// Brief: Slave Arm Run Self-check Trajectory
FUNCTION_BLOCK PUBLIC FB_SlaveCtrlInstruRetract EXTENDS FB_SlaveArmCtrlBase
VAR_INPUT
END_VAR
VAR_OUTPUT
END_VAR
VAR
	m_retractPlanner:FB_BasicDoubleS;;
	
	m_retractVel: LREAL:= 0.05;
	m_retractAcc: LREAL:= 0.1;
	m_retractJerk: LREAL:= 1;
	
	m_retractLimitBuffer:LREAL := 0.02;
	m_retractPos :LREAL;
	
END_VAR

// override this function in each exact controller
METHOD PROTECTED calcCmdJntPos : BOOL
VAR_IN_OUT CONSTANT
	i_endoscopePose : ST_Frame;
	i_masterStatus :ST_MasterStatus;
	i_setupStatus: ST_SetupStatus;
	i_slaveArm :FB_SlaveArm;
END_VAR

VAR 
	i :INT;
	curJntVel :Vec8d;
END_VAR
// check if planner is ready
IF m_retractPlanner.isGene = FALSE THEN
	calcCmdJntPos:=FALSE;
	m_timePeriod:=0;
	RETURN;
END_IF

// traj plan
calcCmdJntPos :=m_retractPlanner.evaluate(m_timePeriod, q=> m_cmdJntPos[3], q_dot=>m_cmdJntVel[3], q_dot=> m_cmdJntAcc[3]);

IF m_timePeriod > m_retractPlanner.duration AND  ABS(i_slaveArm.curJntPos[3] - m_retractPos) < g_cartCtrlPosTolHign THEN
	m_isFinished:=TRUE;
END_IF
END_METHOD

METHOD PUBLIC init : BOOL
VAR_IN_OUT CONSTANT
	i_slaveArm	:FB_SlaveArm;
END_VAR
VAR_IN_OUT 
	r_slaveArmCtrlCmd :ST_SlaveArmCtrlCmds;
END_VAR

VAR
	q:ARRAY[1..2] OF LREAL;
	v:ARRAY[1..2] OF LREAL;
END_VAR
// check if to hold the command joint position unchanged
m_holdLastCmds := checkToHoldLastCmds(i_slaveArm);

SUPER^.Init(i_slaveArm,r_slaveArmCtrlCmd);

// planning for joint3 motion
m_retractPos :=GVL_SlaveMotorParameters.g_maxJntPos[3]+m_retractLimitBuffer;
q[1]:=i_slaveArm.curJntPos[3];
q[2]:= m_retractPos;
v[1]:=0;
v[2]:=0;
m_retractPlanner.init(q,v, m_retractVel, m_retractAcc, m_retractJerk);
END_METHOD

END_FUNCTION_BLOCK

(* stored: Version 1.1.0.1, ProductVersion 3.1.4024.11
   POU FB_SlaveCtrlInstruRetract: Id {596332da-68eb-4244-8a80-7e3d57b3bb9f}, SpecialFunc None
   Method calcCmdJntPos: Id {7b11d094-8bfe-4cb8-971c-9702c727740e}
   Method init: Id {7aae2cb5-3dc8-47a4-84c8-fce1eb91d921} *)
